{attribute 'GeneratedUsingTerminal: CMMP-AS V4p0 CiA402-0002'}
{attribute addProperty BoxType "CMMP-AS V4p0 CiA402-0002"}
{attribute addProperty Id "Velocity_Actual_ValueAT %I*DINT4Following_Error_Actual_ValueAT %I*DINT4"}
{attribute addProperty CRC "2219913602"}
{attribute addProperty Size "8"}
TYPE Inputs_84513182 EXTENDS TcoIo.InputBase_8311D824 :
STRUCT
	{attribute addProperty Name "Velocity_Actual_Value"}
	Velocity_Actual_Value AT %I* : DINT;
	{attribute addProperty Name "Following_Error_Actual_Value"}
	Following_Error_Actual_Value AT %I* : DINT;
END_STRUCT
END_TYPE

(* stored: Version 1.2.0.0, ProductVersion 3.1.4024.11
   DUT Inputs_84513182: Id {0d3affdd-c733-0787-319f-1a51b945e640} *)
